(* IEC 61131-3 sources: AXOpen/src/integrations/app/src, 3 files *)

(* ---- recipe.st ---- *)
{#ix-attr:[Container(Layout.Tabs)]}
{#ix-attr:[Group(GroupLayout.GroupBox)]}
{#ix-set:AttributeName = "This is some structure"}
{S7.extern=ReadWrite}
CLASS PUBLIC Recipe
    VAR PUBLIC
        Header : ReciepeHeader;
        Measurements : Measurements;
        Colors : Colors;
    END_VAR
END_CLASS

TYPE
    Colors : (RED, GREEN, BLUE);
END_TYPE

{#ix-attr:[Container(Layout.Stack)]}
{S7.extern=ReadWrite}
CLASS PUBLIC ReciepeHeader
    VAR PUBLIC
        Name : STRING;
    END_VAR
END_CLASS

{#ix-attr:[Container(Layout.Tabs)]}
{S7.extern=ReadWrite}
CLASS PUBLIC Measurements
    VAR PUBLIC
        {#ix-set:AttributeName = "Dimension X"}
        DimX : ContinuesValueCheckData;
        {#ix-set:AttributeName = "Dimension Y"}
        DimY : ContinuesValueCheckData;
        {#ix-set:AttributeName = "Dimension Z"}
        DimZ : ContinuesValueCheckData;
        {#ix-set:AttributeName = "Inside temp °C"}
        TemperatureIn : ContinuesValueCheckData;
        {#ix-set:AttributeName = "Outside temp °C"}
        TemperatureOut : ContinuesValueCheckData;
    END_VAR
END_CLASS

{#ix-attr:[Container(Layout.Wrap)]}
{#ix-attr:[Group(GroupLayout.GroupBox)]}
{S7.extern=ReadWrite}
CLASS PUBLIC ContinuesValueCheckData
    VAR PUBLIC
        Min : REAL;
        Measured : REAL;
        Max : REAL;
    END_VAR
END_CLASS

(* ---- program.st ---- *)
USING AXOpen.Core;

PROGRAM MyProgram
    VAR_EXTERNAL
        MainContext : MyContext;
        I_am_alive : ULINT;
        AxoSequencers : AxoSequencerExamples.SequencerExample;
        AxoSequencerContainer : AxoSequencerContainerExamples.SequencerContainerExample;
        AxoTasks : AxoTaskExamples.Tasks;
        AxoTaskDocu : AxoTaskExamples.AxoTaskDocuExample;
        myComponentExample : AxoComponentExamples.ComponentExampleContext;
        myComponentHeaderOnlyExample : AxoComponentExamples.ComponentHeaderOnlyExampleContext;
        AxoRemoteTasks : AxoRemoteTaskExamples.RemoteTasks;
        AxoToggleTasks : AxoToggleTaskExamples.Tasks;
        AxoToggleTaskDocu : AxoToggleTaskExamples.AxoToggleTaskDocuExample;
        AxoMomentaryTasks : AxoMomentaryTaskExamples.Tasks;
        AxoMomentaryTaskDocu : AxoMomentaryTaskExamples.AxoMomentaryTaskDocuExample;

        AxoDataExamplesDocu : AxoDataExamplesDocu.Context;

        AxoMessengers : AxoStaticMessengerExample.Messengers;
        AxoMessengersDocu : AxoStaticMessengerDocuExample.Messengers;

        AxoDataFragmentExchangeContext : AxoDataFramentsExchangeDocuExample.AxoDataFragmentExchangeContext;
        AxoTextListExampleContext : AxoTextListExample.AxoTextListExampleContext;
        AxoCognexVisionDatamanExampleContext : AxoCognexVisionDatamanExamples.AxoCognexVisionDatamanExampleContext;
        AxoCognexVisionInsightExampleContext : AxoCognexVisionInsightExamples.AxoCognexVisionInsightExampleContext;
        AxoByteArrayExampleContext : AxoByteArrayExample.AxoByteArrayExampleContext;
        AxoBoolArrayExampleContext : AxoBoolArrayExample.AxoBoolArrayExampleContext;

        AxoLoggers : AxoLoggerExamples.Loggers;

        // Integration test
        Integrations : IntegrationTests.Integrations;
        AxoRtc : AxoRtc.AxoS71500Rtc;

    END_VAR

    I_am_alive := I_am_alive + ULINT#1;

    MainContext.Run();
    AxoTasks.Run();
    AxoTaskDocu.Run();
    AxoToggleTasks.Run();
    AxoToggleTaskDocu.Run();
    AxoSequencers.Run();
    AxoSequencerContainer.Run();
    myComponentExample.Run();
    myComponentHeaderOnlyExample.Run();
    AxoRemoteTasks.Run();
    AxoMomentaryTasks.Run();
    AxoMomentaryTaskDocu.Run();
    AxoDataExamplesDocu.Run();
    AxoMessengers.Run();
    AxoMessengers.InjectRtc(AxoRtc);
    AxoMessengersDocu.Run();
    AxoMessengersDocu.InjectRtc(AxoRtc);
    AxoDataFragmentExchangeContext.Run();

    AxoTextListExampleContext.Run();

    AxoCognexVisionDatamanExampleContext.InjectRtc(AxoRtc);
    AxoCognexVisionDatamanExampleContext.Run();

    AxoCognexVisionInsightExampleContext.InjectRtc(AxoRtc);
    AxoCognexVisionInsightExampleContext.Run();
    AxoByteArrayExampleContext.Run();
    AxoBoolArrayExampleContext.Run();

    AxoLoggers.InjectRtc(AxoRtc);
    AxoLoggers.Run();
    // Integration tests
    Integrations.Run();

END_PROGRAM

{S7.extern=ReadWrite}
CLASS MyContext EXTENDS AxoContext
    VAR PUBLIC
        process_data_manager: AxoDataExamples.AxoProcessDataManager;
        test_data_manager: AxoDataExamples.AxoTestDataManager;
        _rootObject :   AxoObject;
    END_VAR

    METHOD PROTECTED OVERRIDE Main
        THIS.DataExchangeTests();
    END_METHOD

    METHOD DataExchangeTests : Int
        THIS.InitializeRootObject(_rootObject);
        process_data_manager.Run(_rootObject);

        IF(process_data_manager._create) THEN
            IF(process_data_manager.Create(process_data_manager._identifier).IsDone()) THEN
                process_data_manager._create := FALSE;
            END_IF;
        END_IF;

        IF(process_data_manager._read) THEN
            IF(process_data_manager.Read(process_data_manager._identifier).IsDone()) THEN
                process_data_manager._read := FALSE;
            END_IF;
        END_IF;

        IF(process_data_manager._update) THEN
            IF(process_data_manager.Update(process_data_manager._identifier).IsDone()) THEN
                process_data_manager._update := FALSE;
            END_IF;
        END_IF;

        IF(process_data_manager._delete) THEN
            IF(process_data_manager.Delete(process_data_manager._identifier).IsDone()) THEN
                process_data_manager._delete := FALSE;
            END_IF;
        END_IF;
    END_METHOD
END_CLASS

(* ---- configuration.st ---- *)
USING VmT;
CONFIGURATION MyConfiguration
    TASK Main(Interval := T#10ms, Priority := 1);
    PROGRAM P1 WITH Main: MyProgram;
    PROGRAM P2 WITH Main: ProgramExample;

    VAR_GLOBAL
        {#ix-attr:[Container(Layout.Wrap)]}
        {S7.extern=ReadWrite}
        MainContext : MyContext;
        {S7.extern=ReadWrite}
        Recipe : Recipe;
        {#ix-set:AttributeName = "If counting PLC is alive"}
        {S7.extern=ReadWrite}
        I_am_alive : ULINT;
        {S7.extern=ReadWrite}
        AxoSequencers : AxoSequencerExamples.SequencerExample;
        {S7.extern=ReadWrite}
        AxoSequencerContainer : AxoSequencerContainerExamples.SequencerContainerExample;
        {S7.extern=ReadWrite}
        AxoTasks : AxoTaskExamples.Tasks;
        {S7.extern=ReadWrite}
        AxoTaskDocu : AxoTaskExamples.AxoTaskDocuExample;
        {S7.extern=ReadWrite}
        myComponentExample : AxoComponentExamples.ComponentExampleContext;
        {S7.extern=ReadWrite}
        myComponentHeaderOnlyExample : AxoComponentExamples.ComponentHeaderOnlyExampleContext;
        {S7.extern=ReadWrite}
        AxoRemoteTasks : AxoRemoteTaskExamples.RemoteTasks;
        {S7.extern=ReadWrite}
        AxoToggleTasks : AxoToggleTaskExamples.Tasks;
        {S7.extern=ReadWrite}
        AxoToggleTaskDocu : AxoToggleTaskExamples.AxoToggleTaskDocuExample;
        {S7.extern=ReadWrite}
        AxoMomentaryTasks : AxoMomentaryTaskExamples.Tasks;
        {S7.extern=ReadWrite}
        AxoMomentaryTaskDocu : AxoMomentaryTaskExamples.AxoMomentaryTaskDocuExample;
        {S7.extern=ReadWrite}
        AxoDataExamplesDocu : AxoDataExamplesDocu.Context;
        {S7.extern=ReadWrite}
        AxoMessengers : AxoStaticMessengerExample.Messengers;
        {S7.extern=ReadWrite}
        AxoMessengersDocu : AxoStaticMessengerDocuExample.Messengers;
        {S7.extern=ReadWrite}
        AxoRtc : AxoRtc.AxoS71500Rtc;
        {S7.extern=ReadWrite}
        AxoDataFragmentExchangeContext : AxoDataFramentsExchangeDocuExample.AxoDataFragmentExchangeContext;
        {S7.extern=ReadWrite}
        AxoTextListExampleContext : AxoTextListExample.AxoTextListExampleContext;
        {S7.extern=ReadWrite}
        AxoByteArrayExampleContext : AxoByteArrayExample.AxoByteArrayExampleContext;
        {S7.extern=ReadWrite}
        AxoBoolArrayExampleContext : AxoBoolArrayExample.AxoBoolArrayExampleContext;

        {S7.extern=ReadWrite}
        process_data_manager: AxoDataExamples.AxoProcessDataManager;
        {S7.extern=ReadWrite}
        test_data_manager: AxoDataExamples.AxoTestDataManager;
        {S7.extern=ReadWrite}
        AxoLoggers : AxoLoggerExamples.Loggers;
        // Issues
        {S7.extern=ReadWrite}
        gh_ptku_8 : Layouts.Tabbed.weather;

        // Integration tests
        {S7.extern=ReadWrite}
        Integrations : IntegrationTests.Integrations;
    END_VAR

END_CONFIGURATION
